FUNCTION_BLOCK INTERNAL FB_HmiBaseControlTrigger
VAR_INPUT
	stHmiToPlcIn 	: ST_DefaultHmiToPlc;
END_VAR
VAR_IN_OUT
	stHmiToPlcOut 	: ST_DefaultHmiToPlc;
END_VAR
VAR
	fTrigStart	: F_TRIG;
	fTrigStop	: F_TRIG;
	fTrigReset	: F_TRIG;
	fTrigTip	: F_TRIG;
	
	tonHome		: TON;
	rTrigHome	: R_TRIG;
	
	fTrigOpModeManual	: F_TRIG;
	fTrigOpModeAuto		: F_TRIG;
	fTrigOpModeStep		: F_TRIG;
END_VAR

fTrigStart(CLK := stHmiToPlcIn.bStart, Q => stHmiToPlcOut.bStart);
stHmiToPlcOut.bStop := stHmiToPlcIn.bStop;
stHmiToPlcOut.bFastStop := stHmiToPlcIn.bFastStop;
stHmiToPlcOut.eSafetyOpMode := stHmiToPlcIn.eSafetyOpMode;
fTrigReset(CLK := stHmiToPlcIn.bReset, Q => stHmiToPlcOut.bReset);
fTrigTip(CLK := stHmiToPlcIn.bStep, Q => stHmiToPlcOut.bStep);

tonHome(IN := stHmiToPlcIn.bHome, PT := T#1S);
rTrigHome(CLK := tonHome.Q, Q => stHmiToPlcOut.bHome);

fTrigOpModeManual(CLK := stHmiToPlcIn.bOpModeManual, Q => stHmiToPlcOut.bOpModeManual);
fTrigOpModeAuto(CLK := stHmiToPlcIn.bOpModeAuto, Q => stHmiToPlcOut.bOpModeAuto);
fTrigOpModeStep(CLK := stHmiToPlcIn.bOpModeStep, Q => stHmiToPlcOut.bOpModeStep);

END_FUNCTION_BLOCK

(* stored: Version 1.1.0.1, ProductVersion 3.1.4024.12
   POU FB_HmiBaseControlTrigger: Id {694e59bb-6e93-43d1-9d14-86df755e3257}, SpecialFunc None *)
